//EL9505 | Power supply terminal 5V
FUNCTION_BLOCK EL9505

VAR_INPUT
	En: BOOL;
	iTerminal_ID	: INT;
	ErrorSystem		: POINTER TO ST_ErrorSystem;
END_VAR

VAR_OUTPUT
	EnO		: BOOL;
	bError	: BOOL;
END_VAR

VAR
	bUoPwr_OK			AT %I*	: BOOL;
	bUo_Overload		AT %I*	: BOOL;
	WcState_WcState		AT %I*	: BOOL;
	InfoData_State		AT %I*	: UINT;
	
	//FB-s
	EL9505_Error : FB_TerminalError;
	PWR_Error		: FB_GenericError;
END_VAR

(*
* TODO: Test on hardware
*)
EnO:=En;

IF En THEN
	IF 	(NOT bUoPwr_OK) OR bUo_Overload THEN
		PWR_Error.sErrorMessage		:= 'EL9505: ';
		IF NOT bUoPwr_OK	THEN	PWR_Error.sErrorMessage := CONCAT (PWR_Error.sErrorMessage, 'Output Voltage Error; ');		PWR_Error.ErrorPriority := 5;		END_IF
		IF bUo_Overload		THEN	PWR_Error.sErrorMessage := CONCAT (PWR_Error.sErrorMessage, 'Overload; ');					PWR_Error.ErrorPriority := 5;		END_IF
		PWR_Error.bError	:= TRUE;
	ELSE
		PWR_Error.sErrorMessage	:= '';
		PWR_Error.bError		:= FALSE;
	END_IF

END_IF


//Error FB instance
EL9505_Error(
	En := TRUE,
	iTerminal_ID := iTerminal_ID,
	bWcState := WcState_WcState,
	uiInfoData_State := InfoData_State,
	pErrorSystem := ErrorSystem,
	bError => bError,
);

PWR_Error (
	En					:= TRUE,
	bError				:= ,
	sErrorMessage		:= ,
	ErrorPriority		:= ,
	iTerminal_ID		:= iTerminal_ID,
	pErrorSystem		:= ErrorSystem,
	EnO					=> ,
);

END_FUNCTION_BLOCK

(* stored: Version 1.1.0.1, ProductVersion 3.1.4022.17
   POU EL9505: Id {010a0f13-6d5c-4f48-8fc5-897e7583293a}, SpecialFunc None *)
